FUNCTION_BLOCK FB_TataNexon EXTENDS FB_Car

VAR_INPUT
	nNum : INT;
END_VAR
VAR
	bStart : BOOL;
	bDriving : BOOL;
END_VAR

METHOD Drive : BOOL
VAR_INPUT
END_VAR
bDriving := TRUE;
END_METHOD

METHOD  Start : BOOL
VAR_INPUT
END_VAR
bStart := TRUE;
END_METHOD

END_FUNCTION_BLOCK

(* stored: Version 1.1.0.1, ProductVersion 3.1.4024.16
   POU FB_TataNexon: Id {899ab903-5695-4ffe-b13d-79245160d5f3}, SpecialFunc None
   Method Drive: Id {d4b51ee1-4e67-44d0-86ef-49496348bc8c}
   Method Start: Id {e8e18b09-07b4-493b-8fdd-1ae28fb607d3} *)
